FUNCTION_BLOCK StopMoverGroup EXTENDS TaskBase
VAR_INPUT
END_VAR
VAR_OUTPUT
END_VAR
VAR
	groupStop			: MC_GroupStop;
	_caGroup			: ICollisionGroup;
	_stopGroup : BOOL;
	_jerk : MC_LREAL;
	_deceleration : MC_LREAL;
	Logger : TcMessage_Ext;
END_VAR

METHOD Abort : BOOL
groupStop.Execute := FALSE;
State := 0;
Abort := true;
END_METHOD

METHOD Cycle : BOOL
VAR_INPUT
END_VAR
CASE State OF
	0:
		IF _stopGroup THEN
			_done := FALSE;
			_error := FALSE;
			_busy := TRUE;
			groupStop.Execute := TRUE;
			IF groupStop.Busy THEN
				State := 10;
				_stopGroup := FALSE;
				Logger.Send(TC_EVENTS.XtsCAGroupEvents.CAGroupStopping,'');
			END_IF
		END_IF
	10:
		IF groupStop.Done THEN
			_done := TRUE;
			Logger.Send(TC_EVENTS.XtsCAGroupEvents.CAGroupStopped,'');
		ELSIF groupStop.Error THEN
			_error := TRUE;
			Logger.Send(TC_EVENTS.XtsCAGroupEvents.CAGroupStopError,'');
		END_IF
		IF _done OR _error THEN
			_busy := FALSE;
			groupStop.Execute := FALSE;
			State := 0;
		END_IF
END_CASE


groupStop(AxesGroup := _caGroup.GroupRef);
END_METHOD

PROPERTY PUBLIC Deceleration : MC_LREAL
GET
Deceleration := _deceleration;
END_GET
SET
_deceleration := Deceleration;
END_SET
END_PROPERTY

METHOD Execute : BOOL
_stopGroup := Execute := true;
END_METHOD

METHOD FB_init : BOOL
VAR_INPUT
	bInitRetains : BOOL; // if TRUE, the retain variables are initialized (warm start / cold start)
	bInCopyCode : BOOL;  // if TRUE, the instance afterwards gets moved into the copy code (online change)
	CAGroup : ICollisionGroup;
END_VAR
_caGroup := CAGroup;
END_METHOD

PROPERTY PUBLIC Jerk : MC_LREAL
GET
Jerk := _jerk;
END_GET
SET
_jerk := Jerk;
END_SET
END_PROPERTY

END_FUNCTION_BLOCK

(* stored: Version 1.1.0.1, ProductVersion 3.1.4024.12
   POU StopMoverGroup: Id {eb49de9c-c73f-4d5d-a00e-2a61463004b7}, SpecialFunc None
   Method Abort: Id {72cda355-8b53-47d8-a9a5-10a15a81f986}
   Method Cycle: Id {1b69b692-0cbb-4a51-a184-3fdd67c7fdf9}
   Property Deceleration: Id {bfbefcb0-fbdf-4b0b-910d-3a760f3dacc8}
   Get Get: Id {7bce0187-c5f1-4f16-ae78-2053eac6b73a}
   Set Set: Id {b9c66c23-7370-4c93-a332-10bc21b77278}
   Method Execute: Id {47b4c514-d6a1-4abb-9737-014dd8533d0b}
   Method FB_init: Id {011380c3-171f-4a6a-b6fa-f3f46833b181}
   Property Jerk: Id {05c29a4f-80d9-4320-ab90-26b6b39a5d0c}
   Get Get: Id {ddecc54b-81c3-48ab-9470-b3e950a67a9e}
   Set Set: Id {1fad4a9c-0a2e-4c6c-b771-60f32adb2177} *)
